Yaskawa INFORM job: R1-MOVE.JBI

/JOB
//NAME R1-MOVE
//POS
///NPOS 6,0,0,0,0,0
///TOOL 0
///POSTYPE PULSE
///PULSE
C00000=-6744,-46438,-34826,-14046,-21223,6588
C00001=-41249,-46438,-34826,-14046,-21223,6588
C00002=-41249,-46438,-64636,-14046,-21223,6588
C00003=27444,-46438,-64636,-14046,-21223,6588
C00004=27444,-46438,-32335,-14046,-21223,6588
C00005=-9842,-46438,-32335,-14046,-21223,6588
//INST
///DATE 2023/02/06 16:49
///ATTR SC,RW
///GROUP1 RB1
NOP
MOVL C00000 V=83.3
MOVL C00001 V=83.3
MOVL C00002 V=83.3
MOVL C00003 V=83.3
MOVL C00004 V=83.3
MOVL C00005 V=83.3
END
